PROGRAM MAIN
VAR
	XMEAS	: ARRAY[1..41] OF LREAL;
END_VAR

END_PROGRAM

(* stored: Version 1.1.0.1, ProductVersion 3.1.0.36
   POU MAIN: Id {e0a4d229-b224-4048-b09c-d1848ff7d0a0}, SpecialFunc None *)
